// TwinCAT 3 PLC project Sample04
// ProgramVersion: 3.1.4023.0
// libraries:
//   Tc2_Standard, * (Beckhoff Automation GmbH)
//   Tc2_System, * (Beckhoff Automation GmbH)
//   Tc3_Module, * (Beckhoff Automation GmbH)
// project tree:
//   DUTs/ ST_SequenceItem.TcDUT
//   / PlcTask.TcTTO
//   POUs/ Class Diagram.TcCD (not stored), FB_SequenceManager.TcPOU, FB_SequenceSortedByValueAscending.TcPOU, FB_SequenceSortedByValueDescending.TcPOU, FB_SequenceSortedByIdAscending.TcPOU, FB_SequenceSortedByIdDescending.TcPOU, FB_SequenceSortedByDurationAscending.TcPOU, FB_SequenceSortedByDurationDescending.TcPOU, I_SequenceSortable.TcIO, MAIN.TcPOU
// real-time tasks:
//   TASK PlcTask: cycle T#10ms, priority 20, ADS port 350

CONFIGURATION Sample04
    RESOURCE PLC ON TwinCAT3
        TASK PlcTask(INTERVAL := T#10ms, PRIORITY := 20);
        PROGRAM MAIN WITH PlcTask : MAIN;
    END_RESOURCE
END_CONFIGURATION

// ---- DUTs/ST_SequenceItem.TcDUT
TYPE ST_SequenceItem :
STRUCT
	nId			: UINT;
	nValue		: USINT(0..100);
	nDuration	: UINT;
END_STRUCT
END_TYPE

// ---- POUs/I_SequenceSortable.TcIO
INTERFACE I_SequenceSortable EXTENDS __SYSTEM.IQueryInterface

METHOD SortList
VAR_INPUT
	refSequence			: REFERENCE TO ARRAY [1..5] OF ST_SequenceItem;
END_VAR
END_METHOD

END_INTERFACE

// ---- POUs/MAIN.TcPOU
PROGRAM MAIN
VAR
	fbSequenceManager						: FB_SequenceManager;
	fbSequenceSortedByIdAscending			: FB_SequenceSortedByIdAscending;
	fbSequenceSortedByValueAscending		: FB_SequenceSortedByValueAscending;
	fbSequenceSortedByDurationAscending		: FB_SequenceSortedByDurationAscending;
	fbSequenceSortedByIdDescending			: FB_SequenceSortedByIdDescending;
	fbSequenceSortedByValueDescending		: FB_SequenceSortedByValueDescending;
	fbSequenceSortedByDurationDescending	: FB_SequenceSortedByDurationDescending;
	nTest									: INT;
END_VAR

IF (nTest = 1) THEN
	fbSequenceManager.Sort(fbSequenceSortedByIdAscending);
	nTest := 0;
ELSIF (nTest = 2) THEN
	fbSequenceManager.Sort(fbSequenceSortedByValueAscending);
	nTest := 0;
ELSIF (nTest = 3) THEN
	fbSequenceManager.Sort(fbSequenceSortedByDurationAscending);
	nTest := 0;
ELSIF (nTest = 4) THEN
	fbSequenceManager.Sort(fbSequenceSortedByIdDescending);
	nTest := 0;
ELSIF (nTest = 5) THEN
	fbSequenceManager.Sort(fbSequenceSortedByValueDescending);
	nTest := 0;
ELSIF (nTest = 6) THEN
	fbSequenceManager.Sort(fbSequenceSortedByDurationDescending);
	nTest := 0;
END_IF

END_PROGRAM

// ---- POUs/FB_SequenceManager.TcPOU
FUNCTION_BLOCK PUBLIC FB_SequenceManager
VAR_INPUT
END_VAR
VAR_OUTPUT
END_VAR
VAR
	// backing variable
	_aSequence	: ARRAY [1..5] OF ST_SequenceItem := [(nId := 1, nValue := 50, nDuration := 20),
													  (nId := 2, nValue := 10, nDuration := 30),
													  (nId := 3, nValue := 23, nDuration := 10),
													  (nId := 4, nValue := 65, nDuration := 200),
													  (nId := 5, nValue := 45, nDuration := 75)];
END_VAR

{attribute 'monitoring' := 'variable'}
PROPERTY PUBLIC aSequence : ARRAY [1..5] OF ST_SequenceItem
GET
aSequence := _aSequence;
END_GET
END_PROPERTY

METHOD PUBLIC Sort
VAR_INPUT
	ipSequenceSortable		: I_SequenceSortable;
END_VAR
IF (ipSequenceSortable <> 0) THEN
	ipSequenceSortable.SortList(THIS^._aSequence);
END_IF
END_METHOD

END_FUNCTION_BLOCK

// ---- POUs/FB_SequenceSortedByIdAscending.TcPOU
FUNCTION_BLOCK PUBLIC FB_SequenceSortedByIdAscending IMPLEMENTS I_SequenceSortable
VAR_INPUT
END_VAR
VAR_OUTPUT
END_VAR
VAR
END_VAR

METHOD SortList
VAR_INPUT
	refSequence			: REFERENCE TO ARRAY [1..5] OF ST_SequenceItem;
END_VAR
VAR
	stLeft, stRight		: ST_SequenceItem;
	nMax, nIndex		: INT;
	bSwapped			: BOOL;
END_VAR
REPEAT
	bSwapped := FALSE;
	FOR nIndex := 1 TO 4 DO
		stLeft := refSequence[nIndex];
		stRight := refSequence[nIndex + 1];
		IF (stLeft.nId > stRight.nId ) THEN
			refSequence[nIndex + 1] := stLeft;
			refSequence[nIndex] := stRight;
			bSwapped := TRUE;
		END_IF
	END_FOR
UNTIL
	bSwapped = FALSE
END_REPEAT;
END_METHOD

END_FUNCTION_BLOCK

// ---- POUs/FB_SequenceSortedByValueAscending.TcPOU
FUNCTION_BLOCK PUBLIC FB_SequenceSortedByValueAscending IMPLEMENTS I_SequenceSortable
VAR_INPUT
END_VAR
VAR_OUTPUT
END_VAR
VAR
END_VAR

METHOD SortList
VAR_INPUT
	refSequence			: REFERENCE TO ARRAY [1..5] OF ST_SequenceItem;
END_VAR
VAR
	stLeft, stRight		: ST_SequenceItem;
	nMax, nIndex		: INT;
	bSwapped			: BOOL;
END_VAR
REPEAT
	bSwapped := FALSE;
	FOR nIndex := 1 TO 4 DO
		stLeft := refSequence[nIndex];
		stRight := refSequence[nIndex + 1];
		IF (stLeft.nValue > stRight.nValue) THEN
			refSequence[nIndex + 1] := stLeft;
			refSequence[nIndex] := stRight;
			bSwapped := TRUE;
		END_IF
	END_FOR
UNTIL
	bSwapped = FALSE
END_REPEAT;
END_METHOD

END_FUNCTION_BLOCK

// ---- POUs/FB_SequenceSortedByDurationAscending.TcPOU
FUNCTION_BLOCK PUBLIC FB_SequenceSortedByDurationAscending IMPLEMENTS I_SequenceSortable
VAR_INPUT
END_VAR
VAR_OUTPUT
END_VAR
VAR
END_VAR

METHOD SortList
VAR_INPUT
	refSequence			: REFERENCE TO ARRAY [1..5] OF ST_SequenceItem;
END_VAR
VAR
	stLeft, stRight		: ST_SequenceItem;
	nMax, nIndex		: INT;
	bSwapped			: BOOL;
END_VAR
REPEAT
	bSwapped := FALSE;
	FOR nIndex := 1 TO 4 DO
		stLeft := refSequence[nIndex];
		stRight := refSequence[nIndex + 1];
		IF (stLeft.nDuration > stRight.nDuration) THEN
			refSequence[nIndex + 1] := stLeft;
			refSequence[nIndex] := stRight;
			bSwapped := TRUE;
		END_IF
	END_FOR
UNTIL
	bSwapped = FALSE
END_REPEAT;
END_METHOD

END_FUNCTION_BLOCK

// ---- POUs/FB_SequenceSortedByIdDescending.TcPOU
FUNCTION_BLOCK PUBLIC FB_SequenceSortedByIdDescending IMPLEMENTS I_SequenceSortable
VAR_INPUT
END_VAR
VAR_OUTPUT
END_VAR
VAR
END_VAR

METHOD SortList
VAR_INPUT
	refSequence			: REFERENCE TO ARRAY [1..5] OF ST_SequenceItem;
END_VAR
VAR
	stLeft, stRight		: ST_SequenceItem;
	nMax, nIndex		: INT;
	bSwapped			: BOOL;
END_VAR
REPEAT
	bSwapped := FALSE;
	FOR nIndex := 1 TO 4 DO
		stLeft := refSequence[nIndex];
		stRight := refSequence[nIndex + 1];
		IF (stLeft.nId < stRight.nId ) THEN
			refSequence[nIndex + 1] := stLeft;
			refSequence[nIndex] := stRight;
			bSwapped := TRUE;
		END_IF
	END_FOR
UNTIL
	bSwapped = FALSE
END_REPEAT;
END_METHOD

END_FUNCTION_BLOCK

// ---- POUs/FB_SequenceSortedByValueDescending.TcPOU
FUNCTION_BLOCK PUBLIC FB_SequenceSortedByValueDescending IMPLEMENTS I_SequenceSortable
VAR_INPUT
END_VAR
VAR_OUTPUT
END_VAR
VAR
END_VAR

METHOD SortList
VAR_INPUT
	refSequence			: REFERENCE TO ARRAY [1..5] OF ST_SequenceItem;
END_VAR
VAR
	stLeft, stRight		: ST_SequenceItem;
	nMax, nIndex		: INT;
	bSwapped			: BOOL;
END_VAR
REPEAT
	bSwapped := FALSE;
	FOR nIndex := 1 TO 4 DO
		stLeft := refSequence[nIndex];
		stRight := refSequence[nIndex + 1];
		IF (stLeft.nValue < stRight.nValue) THEN
			refSequence[nIndex + 1] := stLeft;
			refSequence[nIndex] := stRight;
			bSwapped := TRUE;
		END_IF
	END_FOR
UNTIL
	bSwapped = FALSE
END_REPEAT;
END_METHOD

END_FUNCTION_BLOCK

// ---- POUs/FB_SequenceSortedByDurationDescending.TcPOU
FUNCTION_BLOCK PUBLIC FB_SequenceSortedByDurationDescending IMPLEMENTS I_SequenceSortable
VAR_INPUT
END_VAR
VAR_OUTPUT
END_VAR
VAR
END_VAR

METHOD SortList
VAR_INPUT
	refSequence			: REFERENCE TO ARRAY [1..5] OF ST_SequenceItem;
END_VAR
VAR
	stLeft, stRight		: ST_SequenceItem;
	nMax, nIndex		: INT;
	bSwapped			: BOOL;
END_VAR
REPEAT
	bSwapped := FALSE;
	FOR nIndex := 1 TO 4 DO
		stLeft := refSequence[nIndex];
		stRight := refSequence[nIndex + 1];
		IF (stLeft.nDuration < stRight.nDuration) THEN
			refSequence[nIndex + 1] := stLeft;
			refSequence[nIndex] := stRight;
			bSwapped := TRUE;
		END_IF
	END_FOR
UNTIL
	bSwapped = FALSE
END_REPEAT;
END_METHOD

END_FUNCTION_BLOCK
